// TIA Portal project "MPS_Measuring" (V16)

(* hardware
DEVICE "S7-1200 station_1"  S7-1200 Station
   slot 0: "Rack_0"  S7-1200 Rack  Rack  V1.0
   slot 1: "PLC_1"  CPU 1214C AC/DC/Rly  6ES7 214-1BG40-0XB0  V4.2
DEVICE "S7-1200 station_2"  S7-1200 Station
   slot 0: "Rack_0"  S7-1200 Rack  Rack  V1.0
   slot 1: "PLC_2"  CPU 1214C AC/DC/Rly  6ES7 214-1BG31-0XB0  V3.0
DEVICE "HMI_1"  KTP600 Basic color PN
   slot 0: "HMI_1"  KTP600 Basic color PN  6AV6 647-0AD11-3AX0  12.0.0.0
   slot 1: "HMI_RT_1"  KTP600 Basic color PN  6AV6 647-0AD11-3AX0  12.0.0.0
   slot 5: "HMI_1.IE_CP_1"  PROFINET Interface  12.0.0.0
      slot 1: "PROFINET Interface_1"  PROFINET Interface
         slot 1: "Port_1"  Port
*)

// ===== PLC "PLC_1"  CPU 1214C AC/DC/Rly =====

VAR_GLOBAL   // PLC tag table "Default tag table"
   "Conveyor_fwd" AT %Q0.0 : Bool;
   "Conveyor_rvs" AT %Q0.1 : Bool;
   "Adv_separator" AT %Q0.2 : Bool;
   "Stopper_On" AT %Q0.3 : Bool;
   "Open_Gripper" AT %Q0.4 : Bool;
   "Gripper_dws" AT %Q0.5 : Bool;
   "Swivel_to_msg" AT %Q0.6 : Bool;
   "wp_beg" AT %I0.0 : Bool;
   "wp_mid" AT %I0.1 : Bool;
   "no_wp_end" AT %I0.2 : Bool;
   "Gripper_open" AT %I0.4 : Bool;
   "Gripper_raised" AT %I0.5 : Bool;
   "Swivel_at_conv" AT %I0.6 : Bool;
   "Swivel_at_msg" AT %I0.7 : Bool;
   "Analog_In" AT %IW64 : Int;
   "wp_measure" AT %MD1 : Real;
   "wp_measured" AT %M0.1 : Bool;   // Workpiece has been measured
   "has_cap" AT %M0.2 : Bool;
   "wp_at_conv" AT %M0.3 : Bool;
   "wp_at_msg" AT %M0.4 : Bool;
END_VAR

// folder: System blocks/Program resources

DATA_BLOCK "IEC_Timer_0_DB"   // DB1
{ S7_Optimized_Access := 'TRUE' }
AUTHOR : Simatic
FAMILY : IEC
NAME : IEC_TMR
VERSION : 1.0
// stored: InstanceOfName IEC_TIMER
"IEC_TIMER"
BEGIN
END_DATA_BLOCK

DATA_BLOCK "IEC_Timer_0_DB_1"   // DB2
{ S7_Optimized_Access := 'TRUE' }
AUTHOR : Simatic
FAMILY : IEC
NAME : IEC_TMR
VERSION : 1.0
// stored: InstanceOfName IEC_TIMER
"IEC_TIMER"
BEGIN
END_DATA_BLOCK

DATA_BLOCK "IEC_Timer_0_DB_2"   // DB3
{ S7_Optimized_Access := 'TRUE' }
AUTHOR : Simatic
FAMILY : IEC
NAME : IEC_TMR
VERSION : 1.0
// stored: InstanceOfName IEC_TIMER
"IEC_TIMER"
BEGIN
END_DATA_BLOCK

DATA_BLOCK "IEC_Timer_0_DB_3"   // DB4
{ S7_Optimized_Access := 'TRUE' }
AUTHOR : Simatic
FAMILY : IEC
NAME : IEC_TMR
VERSION : 1.0
// stored: InstanceOfName IEC_TIMER
"IEC_TIMER"
BEGIN
END_DATA_BLOCK

// folder: (top level)

FUNCTION "Read_Analog_Input" : Void   // FC1, LAD
{ S7_Optimized_Access := 'TRUE' }
VERSION : 0.1
   VAR_INPUT
      Input_channel : Int;
      Lower_value : Int;
      Upper_value : Int;
   END_VAR
   VAR_OUTPUT
      Measure : Real;
   END_VAR
   VAR_TEMP
      Temp1 : Real;
   END_VAR
BEGIN

REGION Network 1
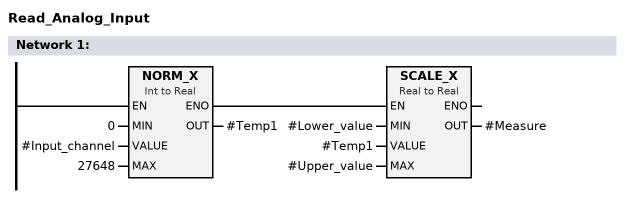
   RUNG wire#powerrail
      { S7_Templates := "[SrcType := Int, DestType := Real]"; S7_GenerateENO := "TRUE" } Normalize(min := 0, value := #Input_channel, max := 27648, out => #Temp1)
      { S7_Templates := "[SrcType := Real, DestType := Real]"; S7_GenerateENO := "TRUE" } Scale(min := #Lower_value, value := #Temp1, max := #Upper_value, out => #Measure)
   END_RUNG
   // the same network as SCL:
   // ENO of a box is taken as its EN; it also drops when the box reports an error
   #Temp1 := NORM_X(MIN := 0, VALUE := #Input_channel, MAX := 27648);
   #Measure := SCALE_X(MIN := #Lower_value, VALUE := #Temp1, MAX := #Upper_value);
END_REGION
END_FUNCTION

FUNCTION "is_capped" : Void   // FC4, LAD
{ S7_Optimized_Access := 'TRUE' }
VERSION : 0.1
   VAR_INPUT
      input_channel : Int;
   END_VAR
   VAR_OUTPUT
      with_cap : Bool;
   END_VAR
   VAR_TEMP
      temp1 : Real;
   END_VAR
   VAR CONSTANT
      cap_det : Real := 0.5;
   END_VAR
   VAR_TEMP   // added for the SCL form of the ladder/FBD networks
      _w1 : Bool;
   END_VAR
BEGIN

REGION Network 1
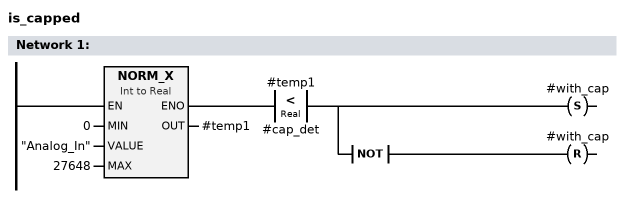
   RUNG wire#powerrail
      { S7_Templates := "[SrcType := Int, DestType := Real]"; S7_GenerateENO := "TRUE" } Normalize(min := 0, value := "Analog_In", max := 27648, out => #temp1)
      { S7_Templates := "SrcType := Real" } LT_Contact(in1 := #temp1, in2 := #cap_det)
      wire#w1
      S_Coil( #with_cap )
   END_RUNG
   RUNG wire#w1
      Not()
      R_Coil( #with_cap )
   END_RUNG
   // the same network as SCL:
   // ENO of a box is taken as its EN; it also drops when the box reports an error
   #temp1 := NORM_X(MIN := 0, VALUE := "Analog_In", MAX := 27648);
   #_w1 := #temp1 < #cap_det;
   IF #_w1 THEN #with_cap := TRUE; END_IF;
   IF NOT #_w1 THEN #with_cap := FALSE; END_IF;
END_REGION
END_FUNCTION

ORGANIZATION_BLOCK "Main"   // OB1, LAD, ProgramCycle
TITLE = "Main Program Sweep (Cycle)"
{ S7_Optimized_Access := 'TRUE' }
VERSION : 0.1
   VAR_TEMP   // added for the SCL form of the ladder/FBD networks
      _w1 : Bool;
   END_VAR
BEGIN

REGION Network 1: Workpiece has been measured
   // Read Measurement
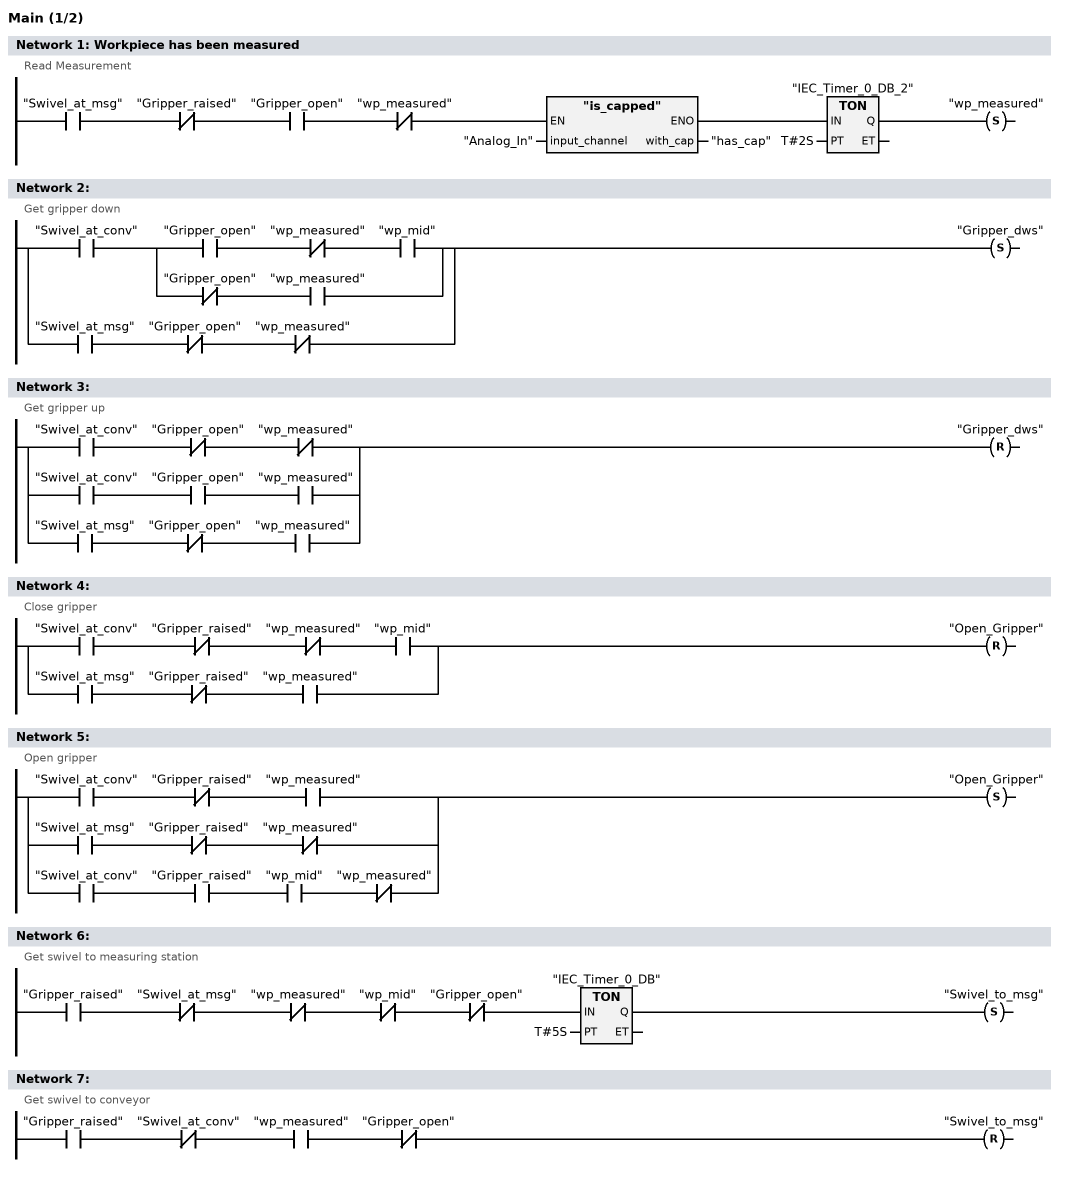
   "is_capped"(EN := "Swivel_at_msg" AND NOT "Gripper_raised" AND "Gripper_open" AND NOT "wp_measured",
               input_channel := "Analog_In",
               with_cap => "has_cap",
               ENO => #_w1);
   "IEC_Timer_0_DB_2".TON(IN := #_w1, PT := T#2S);
   IF "IEC_Timer_0_DB_2".Q THEN "wp_measured" := TRUE; END_IF;
END_REGION

REGION Network 2
   // Get gripper down
   RUNG wire#powerrail
      Contact( "Swivel_at_conv" )
      wire#w1
      Contact( "Gripper_open" )
      I_Contact( "wp_measured" )
      Contact( "wp_mid" )
      wire#w2
      S_Coil( "Gripper_dws" )
   END_RUNG
   RUNG wire#w1
      I_Contact( "Gripper_open" )
      Contact( "wp_measured" )
   END_RUNG wire#w2
   RUNG wire#powerrail
      Contact( "Swivel_at_msg" )
      I_Contact( "Gripper_open" )
      I_Contact( "wp_measured" )
   END_RUNG wire#w2
   // the same network as SCL:
   IF ("Swivel_at_conv" AND (("Gripper_open" AND NOT "wp_measured" AND "wp_mid") OR (NOT "Gripper_open" AND "wp_measured"))) OR ("Swivel_at_msg" AND NOT "Gripper_open" AND NOT "wp_measured") THEN
       "Gripper_dws" := TRUE;
   END_IF;
END_REGION

REGION Network 3
   // Get gripper up
   RUNG wire#powerrail
      Contact( "Swivel_at_conv" )
      I_Contact( "Gripper_open" )
      I_Contact( "wp_measured" )
      wire#w1
      R_Coil( "Gripper_dws" )
   END_RUNG
   RUNG wire#powerrail
      Contact( "Swivel_at_conv" )
      Contact( "Gripper_open" )
      Contact( "wp_measured" )
   END_RUNG wire#w1
   RUNG wire#powerrail
      Contact( "Swivel_at_msg" )
      I_Contact( "Gripper_open" )
      Contact( "wp_measured" )
   END_RUNG wire#w1
   // the same network as SCL:
   IF ("Swivel_at_conv" AND NOT "Gripper_open" AND NOT "wp_measured") OR ("Swivel_at_conv" AND "Gripper_open" AND "wp_measured") OR ("Swivel_at_msg" AND NOT "Gripper_open" AND "wp_measured") THEN
       "Gripper_dws" := FALSE;
   END_IF;
END_REGION

REGION Network 4
   // Close gripper
   RUNG wire#powerrail
      Contact( "Swivel_at_conv" )
      I_Contact( "Gripper_raised" )
      I_Contact( "wp_measured" )
      Contact( "wp_mid" )
      wire#w1
      R_Coil( "Open_Gripper" )
   END_RUNG
   RUNG wire#powerrail
      Contact( "Swivel_at_msg" )
      I_Contact( "Gripper_raised" )
      Contact( "wp_measured" )
   END_RUNG wire#w1
   // the same network as SCL:
   IF ("Swivel_at_conv" AND NOT "Gripper_raised" AND NOT "wp_measured" AND "wp_mid") OR ("Swivel_at_msg" AND NOT "Gripper_raised" AND "wp_measured") THEN
       "Open_Gripper" := FALSE;
   END_IF;
END_REGION

REGION Network 5
   // Open gripper
   RUNG wire#powerrail
      Contact( "Swivel_at_conv" )
      I_Contact( "Gripper_raised" )
      Contact( "wp_measured" )
      wire#w1
      S_Coil( "Open_Gripper" )
   END_RUNG
   RUNG wire#powerrail
      Contact( "Swivel_at_msg" )
      I_Contact( "Gripper_raised" )
      I_Contact( "wp_measured" )
   END_RUNG wire#w1
   RUNG wire#powerrail
      Contact( "Swivel_at_conv" )
      Contact( "Gripper_raised" )
      Contact( "wp_mid" )
      I_Contact( "wp_measured" )
   END_RUNG wire#w1
   // the same network as SCL:
   IF ("Swivel_at_conv" AND NOT "Gripper_raised" AND "wp_measured") OR ("Swivel_at_msg" AND NOT "Gripper_raised" AND NOT "wp_measured") OR ("Swivel_at_conv" AND "Gripper_raised" AND "wp_mid" AND NOT "wp_measured") THEN
       "Open_Gripper" := TRUE;
   END_IF;
END_REGION

REGION Network 6
   // Get swivel to measuring station
   "IEC_Timer_0_DB".TON(IN := "Gripper_raised" AND NOT "Swivel_at_msg" AND NOT "wp_measured" AND NOT "wp_mid" AND NOT "Gripper_open",
                        PT := T#5S);
   IF "IEC_Timer_0_DB".Q THEN "Swivel_to_msg" := TRUE; END_IF;
END_REGION

REGION Network 7
   // Get swivel to conveyor
   RUNG wire#powerrail
      Contact( "Gripper_raised" )
      I_Contact( "Swivel_at_conv" )
      Contact( "wp_measured" )
      I_Contact( "Gripper_open" )
      R_Coil( "Swivel_to_msg" )
   END_RUNG
   // the same network as SCL:
   IF "Gripper_raised" AND NOT "Swivel_at_conv" AND "wp_measured" AND NOT "Gripper_open" THEN
       "Swivel_to_msg" := FALSE;
   END_IF;
END_REGION

REGION Network 8
   // Advance separator
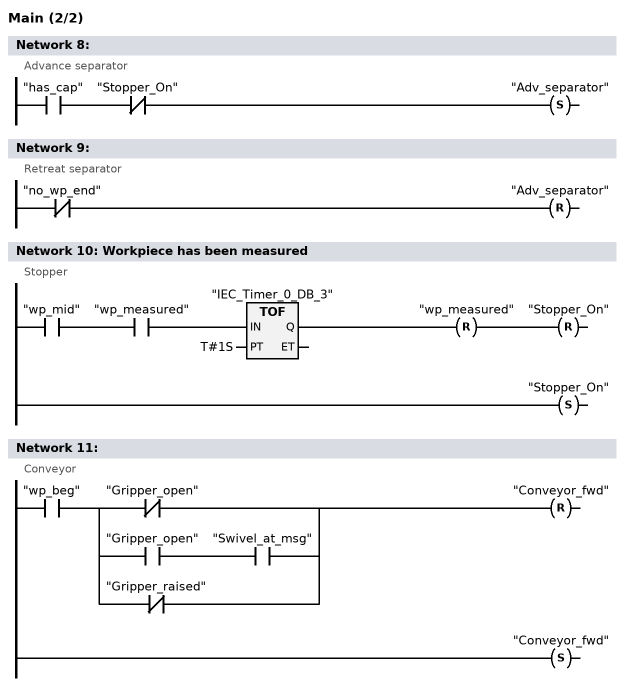
   RUNG wire#powerrail
      Contact( "has_cap" )
      I_Contact( "Stopper_On" )
      S_Coil( "Adv_separator" )
   END_RUNG
   // the same network as SCL:
   IF "has_cap" AND NOT "Stopper_On" THEN "Adv_separator" := TRUE; END_IF;
END_REGION

REGION Network 9
   // Retreat separator
   RUNG wire#powerrail
      I_Contact( "no_wp_end" )
      R_Coil( "Adv_separator" )
   END_RUNG
   // the same network as SCL:
   IF NOT "no_wp_end" THEN "Adv_separator" := FALSE; END_IF;
END_REGION

REGION Network 10: Workpiece has been measured
   // Stopper
   "IEC_Timer_0_DB_3".TOF(IN := "wp_mid" AND "wp_measured", PT := T#1S);
   IF "IEC_Timer_0_DB_3".Q THEN
       "wp_measured" := FALSE;
       "Stopper_On" := FALSE;
   END_IF;
   "Stopper_On" := TRUE;
END_REGION

REGION Network 11
   // Conveyor
   RUNG wire#powerrail
      Contact( "wp_beg" )
      wire#w1
      I_Contact( "Gripper_open" )
      wire#w2
      R_Coil( "Conveyor_fwd" )
   END_RUNG
   RUNG wire#w1
      Contact( "Gripper_open" )
      Contact( "Swivel_at_msg" )
   END_RUNG wire#w2
   RUNG wire#w1
      I_Contact( "Gripper_raised" )
   END_RUNG wire#w2
   RUNG wire#powerrail
      S_Coil( "Conveyor_fwd" )
   END_RUNG
   // the same network as SCL:
   IF "wp_beg" AND (NOT "Gripper_open" OR ("Gripper_open" AND "Swivel_at_msg") OR NOT "Gripper_raised") THEN
       "Conveyor_fwd" := FALSE;
   END_IF;
   "Conveyor_fwd" := TRUE;
END_REGION
END_ORGANIZATION_BLOCK

ORGANIZATION_BLOCK "Startup"   // OB100, LAD, Startup
TITLE = "Complete Restart"
{ S7_Optimized_Access := 'TRUE' }
VERSION : 0.1
   VAR_INPUT
      LostRetentive : Bool;   // True if retentive data are lost
      LostRTC : Bool;   // True if date and time are lost
   END_VAR
BEGIN

REGION Network 1
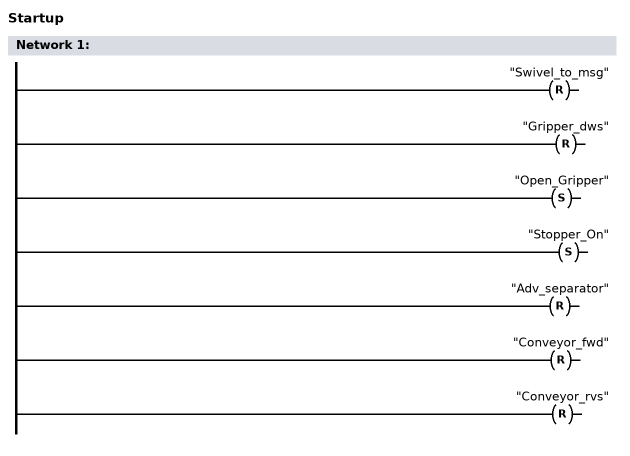
   RUNG wire#powerrail
      R_Coil( "Swivel_to_msg" )
   END_RUNG
   RUNG wire#powerrail
      R_Coil( "Gripper_dws" )
   END_RUNG
   RUNG wire#powerrail
      S_Coil( "Open_Gripper" )
   END_RUNG
   RUNG wire#powerrail
      S_Coil( "Stopper_On" )
   END_RUNG
   RUNG wire#powerrail
      R_Coil( "Adv_separator" )
   END_RUNG
   RUNG wire#powerrail
      R_Coil( "Conveyor_fwd" )
   END_RUNG
   RUNG wire#powerrail
      R_Coil( "Conveyor_rvs" )
   END_RUNG
   // the same network as SCL:
   "Swivel_to_msg" := FALSE;
   "Gripper_dws" := FALSE;
   "Open_Gripper" := TRUE;
   "Stopper_On" := TRUE;
   "Adv_separator" := FALSE;
   "Conveyor_fwd" := FALSE;
   "Conveyor_rvs" := FALSE;
END_REGION
END_ORGANIZATION_BLOCK

// ===== PLC "PLC_2"  CPU 1214C AC/DC/Rly =====

VAR_GLOBAL   // PLC tag table "Default tag table_1"
   "Conveyor_fwd" AT %Q0.0 : Bool;
   "Conveyor_rvs" AT %Q0.1 : Bool;
   "Adv_separator" AT %Q0.2 : Bool;
   "Retract_stopper" AT %Q0.3 : Bool;
   "Open_Gripper" AT %Q0.4 : Bool;
   "Gripper_dws" AT %Q0.5 : Bool;
   "Swivel_to_msg" AT %Q0.6 : Bool;
   "wp_beg" AT %I0.0 : Bool;
   "wp_mid" AT %I0.1 : Bool;
   "no_wp_end" AT %I0.2 : Bool;
   "Gripper_open" AT %I0.6 : Bool;
   "Gripper_raised" AT %I0.5 : Bool;
   "Swivel_at_conv" AT %I0.4 : Bool;
   "Swivel_at_msg" AT %I0.7 : Bool;
   "Analog_In" AT %IW64 : Int;
   "wp_measure" AT %MD1 : Real;
   "wp_measured" AT %M0.1 : Bool;   // Workpiece has been measured
   "has_cap" AT %M0.2 : Bool;
   "wp_at_conv" AT %M0.3 : Bool;
   "wp_at_msg" AT %M0.4 : Bool;
   "stopper_shall_retract" AT %M0.5 : Bool;
   "conv_shall_adv" AT %M0.6 : Bool;
   "system_ready" AT %M0.7 : Bool;
   "reset" AT %M5.0 : Bool;
END_VAR

VAR_GLOBAL CONSTANT   // PLC tag table "Default tag table_1"
   "Local~PROFINET_interface_1~Port_1(1)" : Hw_Interface := 65;
   "OB_Main(1)" : OB_PCYCLE := 1;
   "OB_Startup" : OB_STARTUP := 100;
   "Local(1)" : Hw_SubModule := 49;
   "Local~DI_14_DQ_10_1(1)" : Hw_SubModule := 264;
   "Local~AI_2_1(1)" : Hw_SubModule := 263;
   "Local~MC" : Hw_SubModule := 51;
   "Local~Common" : Hw_SubModule := 50;
   "Local~Device" : Hw_Device := 32;
   "Local~Configuration" : Hw_SubModule := 33;
   "Local~Exec" : Hw_SubModule := 52;
   "Local~HSC_1(1)" : Hw_Hsc := 257;
   "Local~HSC_2(1)" : Hw_Hsc := 258;
   "Local~HSC_3(1)" : Hw_Hsc := 259;
   "Local~HSC_4(1)" : Hw_Hsc := 260;
   "Local~HSC_5(1)" : Hw_Hsc := 261;
   "Local~HSC_6(1)" : Hw_Hsc := 262;
   "Local~Pulse_1(1)" : Hw_Pwm := 265;
   "Local~Pulse_2(1)" : Hw_Pwm := 266;
   "Local~Pulse_3(1)" : Hw_Pwm := 267;
   "Local~Pulse_4(1)" : Hw_Pwm := 268;
   "Local~PROFINET_interface_1(1)" : Hw_Interface := 64;
   "None" : Pip := 65535;
   "Automatic update" : Pip := 0;
   "PIP 1" : Pip := 1;
   "PIP 2" : Pip := 2;
   "PIP 3" : Pip := 3;
   "PIP 4" : Pip := 4;
   "PIP OB Servo" : Pip := 32768;
END_VAR

// folder: System blocks/Program resources

DATA_BLOCK "IEC_Timer_0_DB"   // DB1
{ S7_Optimized_Access := 'TRUE' }
AUTHOR : Simatic
FAMILY : IEC
NAME : IEC_TMR
VERSION : 1.0
// stored: InstanceOfName IEC_TIMER
"IEC_TIMER"
BEGIN
END_DATA_BLOCK

DATA_BLOCK "IEC_Timer_0_DB_1"   // DB2
{ S7_Optimized_Access := 'TRUE' }
AUTHOR : Simatic
FAMILY : IEC
NAME : IEC_TMR
VERSION : 1.0
// stored: InstanceOfName IEC_TIMER
"IEC_TIMER"
BEGIN
END_DATA_BLOCK

DATA_BLOCK "IEC_Timer_0_DB_2"   // DB3
{ S7_Optimized_Access := 'TRUE' }
AUTHOR : Simatic
FAMILY : IEC
NAME : IEC_TMR
VERSION : 1.0
// stored: InstanceOfName IEC_TIMER
"IEC_TIMER"
BEGIN
END_DATA_BLOCK

DATA_BLOCK "IEC_Timer_0_DB_3"   // DB4
{ S7_Optimized_Access := 'TRUE' }
AUTHOR : Simatic
FAMILY : IEC
NAME : IEC_TMR
VERSION : 1.0
// stored: InstanceOfName IEC_TIMER
"IEC_TIMER"
BEGIN
END_DATA_BLOCK

DATA_BLOCK "IEC_Timer_0_DB_4"   // DB5
{ S7_Optimized_Access := 'TRUE' }
AUTHOR : Simatic
FAMILY : IEC
NAME : IEC_TMR
VERSION : 1.0
// stored: InstanceOfName IEC_TIMER
"IEC_TIMER"
BEGIN
END_DATA_BLOCK

DATA_BLOCK "IEC_Timer_0_DB_5"   // DB6
{ S7_Optimized_Access := 'TRUE' }
AUTHOR : Simatic
FAMILY : IEC
NAME : IEC_TMR
VERSION : 1.0
// stored: InstanceOfName IEC_TIMER
"IEC_TIMER"
BEGIN
END_DATA_BLOCK

DATA_BLOCK "IEC_Timer_0_DB_6"   // DB7
{ S7_Optimized_Access := 'TRUE' }
AUTHOR : Simatic
FAMILY : IEC
NAME : IEC_TMR
VERSION : 1.0
// stored: InstanceOfName IEC_TIMER
"IEC_TIMER"
BEGIN
END_DATA_BLOCK

DATA_BLOCK "IEC_Timer_0_DB_7"   // DB8
{ S7_Optimized_Access := 'TRUE' }
AUTHOR : Simatic
FAMILY : IEC
NAME : IEC_TMR
VERSION : 1.0
// stored: InstanceOfName IEC_TIMER
"IEC_TIMER"
BEGIN
END_DATA_BLOCK

DATA_BLOCK "IEC_Timer_0_DB_8"   // DB9
{ S7_Optimized_Access := 'TRUE' }
AUTHOR : Simatic
FAMILY : IEC
NAME : IEC_TMR
VERSION : 1.0
// stored: InstanceOfName IEC_TIMER
"IEC_TIMER"
BEGIN
END_DATA_BLOCK

DATA_BLOCK "IEC_Timer_0_DB_9"   // DB10
{ S7_Optimized_Access := 'TRUE' }
AUTHOR : Simatic
FAMILY : IEC
NAME : IEC_TMR
VERSION : 1.0
// stored: InstanceOfName IEC_TIMER
"IEC_TIMER"
BEGIN
END_DATA_BLOCK

// folder: (top level)

FUNCTION "reset_block" : Void   // FC1, LAD
{ S7_Optimized_Access := 'TRUE' }
VERSION : 0.1
BEGIN

REGION Network 1
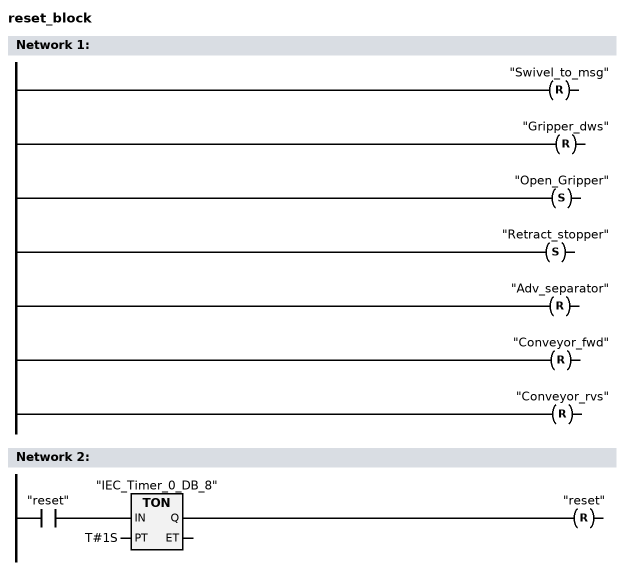
   RUNG wire#powerrail
      R_Coil( "Swivel_to_msg" )
   END_RUNG
   RUNG wire#powerrail
      R_Coil( "Gripper_dws" )
   END_RUNG
   RUNG wire#powerrail
      S_Coil( "Open_Gripper" )
   END_RUNG
   RUNG wire#powerrail
      S_Coil( "Retract_stopper" )
   END_RUNG
   RUNG wire#powerrail
      R_Coil( "Adv_separator" )
   END_RUNG
   RUNG wire#powerrail
      R_Coil( "Conveyor_fwd" )
   END_RUNG
   RUNG wire#powerrail
      R_Coil( "Conveyor_rvs" )
   END_RUNG
   // the same network as SCL:
   "Swivel_to_msg" := FALSE;
   "Gripper_dws" := FALSE;
   "Open_Gripper" := TRUE;
   "Retract_stopper" := TRUE;
   "Adv_separator" := FALSE;
   "Conveyor_fwd" := FALSE;
   "Conveyor_rvs" := FALSE;
END_REGION

REGION Network 2
   "IEC_Timer_0_DB_8".TON(IN := "reset", PT := T#1S);
   IF "IEC_Timer_0_DB_8".Q THEN "reset" := FALSE; END_IF;
END_REGION
END_FUNCTION

FUNCTION "is_capped" : Void   // FC4, LAD
{ S7_Optimized_Access := 'TRUE' }
VERSION : 0.1
   VAR_INPUT
      input_channel : Int;
   END_VAR
   VAR_OUTPUT
      with_cap : Bool;
   END_VAR
   VAR_TEMP
      temp1 : Real;
   END_VAR
   VAR CONSTANT
      cap_det : Real := 0.2;
   END_VAR
   VAR_TEMP   // added for the SCL form of the ladder/FBD networks
      _w1 : Bool;
   END_VAR
BEGIN

REGION Network 1
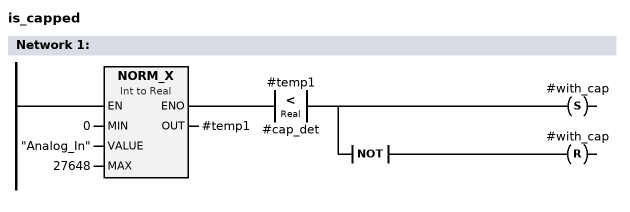
   RUNG wire#powerrail
      { S7_Templates := "[SrcType := Int, DestType := Real]"; S7_GenerateENO := "TRUE" } Normalize(min := 0, value := "Analog_In", max := 27648, out => #temp1)
      { S7_Templates := "SrcType := Real" } LT_Contact(in1 := #temp1, in2 := #cap_det)
      wire#w1
      S_Coil( #with_cap )
   END_RUNG
   RUNG wire#w1
      Not()
      R_Coil( #with_cap )
   END_RUNG
   // the same network as SCL:
   // ENO of a box is taken as its EN; it also drops when the box reports an error
   #temp1 := NORM_X(MIN := 0, VALUE := "Analog_In", MAX := 27648);
   #_w1 := #temp1 < #cap_det;
   IF #_w1 THEN #with_cap := TRUE; END_IF;
   IF NOT #_w1 THEN #with_cap := FALSE; END_IF;
END_REGION
END_FUNCTION

ORGANIZATION_BLOCK "Main"   // OB1, LAD, ProgramCycle
TITLE = "Main Program Sweep (Cycle)"
{ S7_Optimized_Access := 'TRUE' }
VERSION : 0.1
   VAR_TEMP   // added for the SCL form of the ladder/FBD networks
      _w1 : Bool;
      _w2 : Bool;
   END_VAR
BEGIN

REGION Network 1: Workpiece has been measured
   // Read Measurement
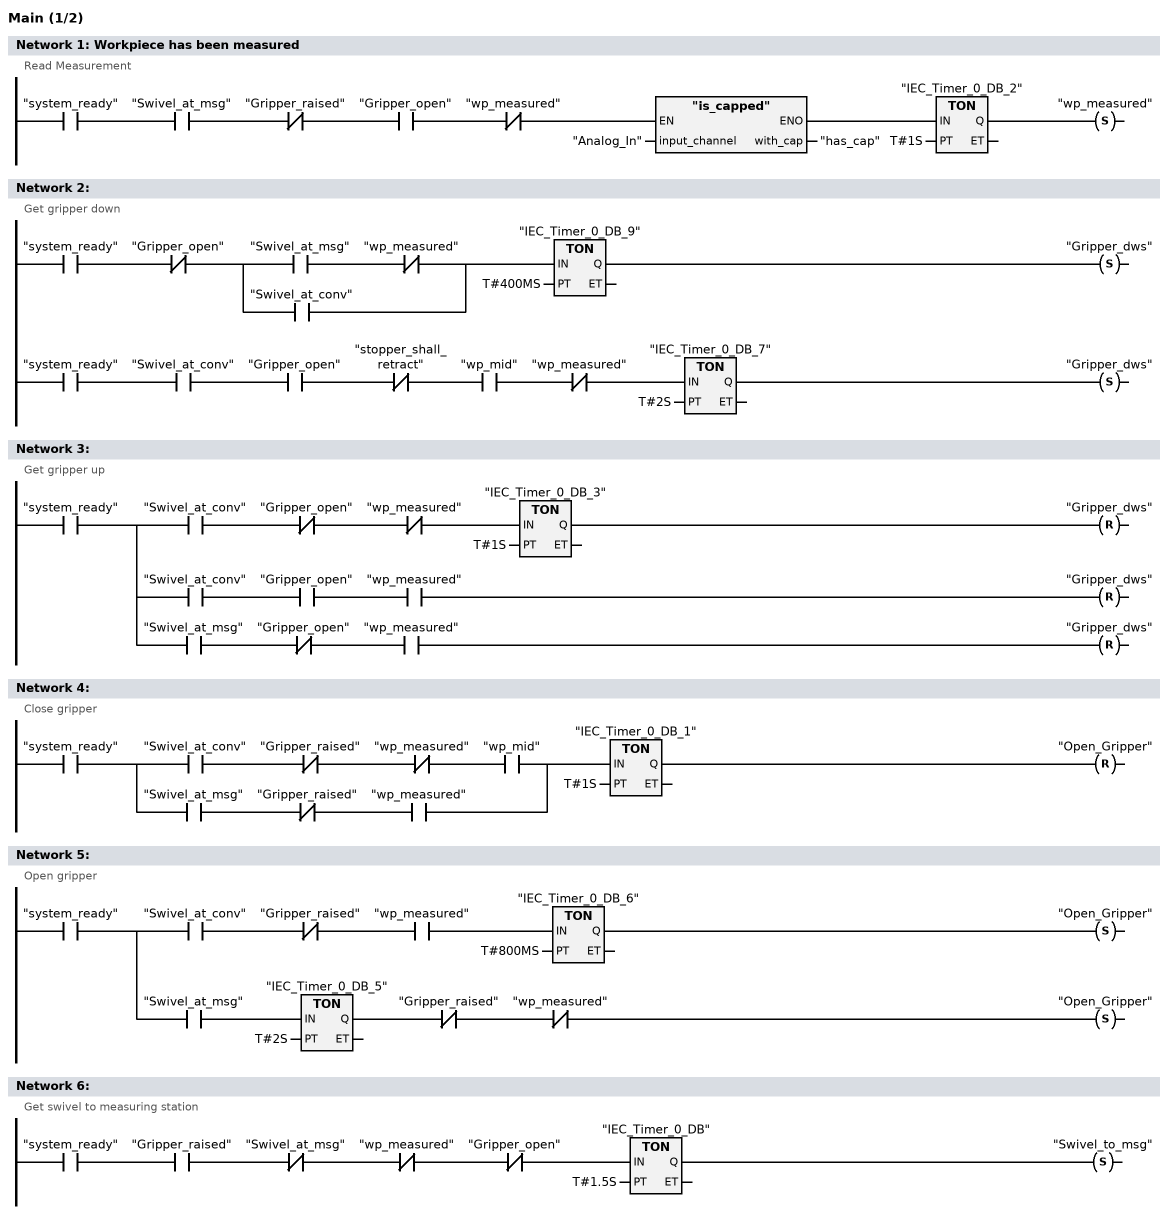
   "is_capped"(EN := "system_ready" AND "Swivel_at_msg" AND NOT "Gripper_raised" AND "Gripper_open" AND NOT "wp_measured",
               input_channel := "Analog_In",
               with_cap => "has_cap",
               ENO => #_w1);
   "IEC_Timer_0_DB_2".TON(IN := #_w1, PT := T#1S);
   IF "IEC_Timer_0_DB_2".Q THEN "wp_measured" := TRUE; END_IF;
END_REGION

REGION Network 2
   // Get gripper down
   "IEC_Timer_0_DB_9".TON(IN := "system_ready" AND NOT "Gripper_open" AND (("Swivel_at_msg" AND NOT "wp_measured") OR "Swivel_at_conv"),
                          PT := T#400MS);
   IF "IEC_Timer_0_DB_9".Q THEN "Gripper_dws" := TRUE; END_IF;
   "IEC_Timer_0_DB_7".TON(IN := "system_ready" AND "Swivel_at_conv" AND "Gripper_open" AND NOT "stopper_shall_retract" AND "wp_mid" AND NOT "wp_measured",
                          PT := T#2S);
   IF "IEC_Timer_0_DB_7".Q THEN "Gripper_dws" := TRUE; END_IF;
END_REGION

REGION Network 3
   // Get gripper up
   "IEC_Timer_0_DB_3".TON(IN := "system_ready" AND "Swivel_at_conv" AND NOT "Gripper_open" AND NOT "wp_measured",
                          PT := T#1S);
   IF "IEC_Timer_0_DB_3".Q THEN "Gripper_dws" := FALSE; END_IF;
   IF "system_ready" AND "Swivel_at_conv" AND "Gripper_open" AND "wp_measured" THEN
       "Gripper_dws" := FALSE;
   END_IF;
   IF "system_ready" AND "Swivel_at_msg" AND NOT "Gripper_open" AND "wp_measured" THEN
       "Gripper_dws" := FALSE;
   END_IF;
END_REGION

REGION Network 4
   // Close gripper
   "IEC_Timer_0_DB_1".TON(IN := "system_ready" AND (("Swivel_at_conv" AND NOT "Gripper_raised" AND NOT "wp_measured" AND "wp_mid") OR ("Swivel_at_msg" AND NOT "Gripper_raised" AND "wp_measured")),
                          PT := T#1S);
   IF "IEC_Timer_0_DB_1".Q THEN "Open_Gripper" := FALSE; END_IF;
END_REGION

REGION Network 5
   // Open gripper
   "IEC_Timer_0_DB_6".TON(IN := "system_ready" AND "Swivel_at_conv" AND NOT "Gripper_raised" AND "wp_measured",
                          PT := T#800MS);
   IF "IEC_Timer_0_DB_6".Q THEN "Open_Gripper" := TRUE; END_IF;
   "IEC_Timer_0_DB_5".TON(IN := "system_ready" AND "Swivel_at_msg", PT := T#2S);
   IF "IEC_Timer_0_DB_5".Q AND NOT "Gripper_raised" AND NOT "wp_measured" THEN
       "Open_Gripper" := TRUE;
   END_IF;
END_REGION

REGION Network 6
   // Get swivel to measuring station
   "IEC_Timer_0_DB".TON(IN := "system_ready" AND "Gripper_raised" AND NOT "Swivel_at_msg" AND NOT "wp_measured" AND NOT "Gripper_open",
                        PT := T#1.5S);
   IF "IEC_Timer_0_DB".Q THEN "Swivel_to_msg" := TRUE; END_IF;
END_REGION

REGION Network 7
   // Get swivel to conveyor
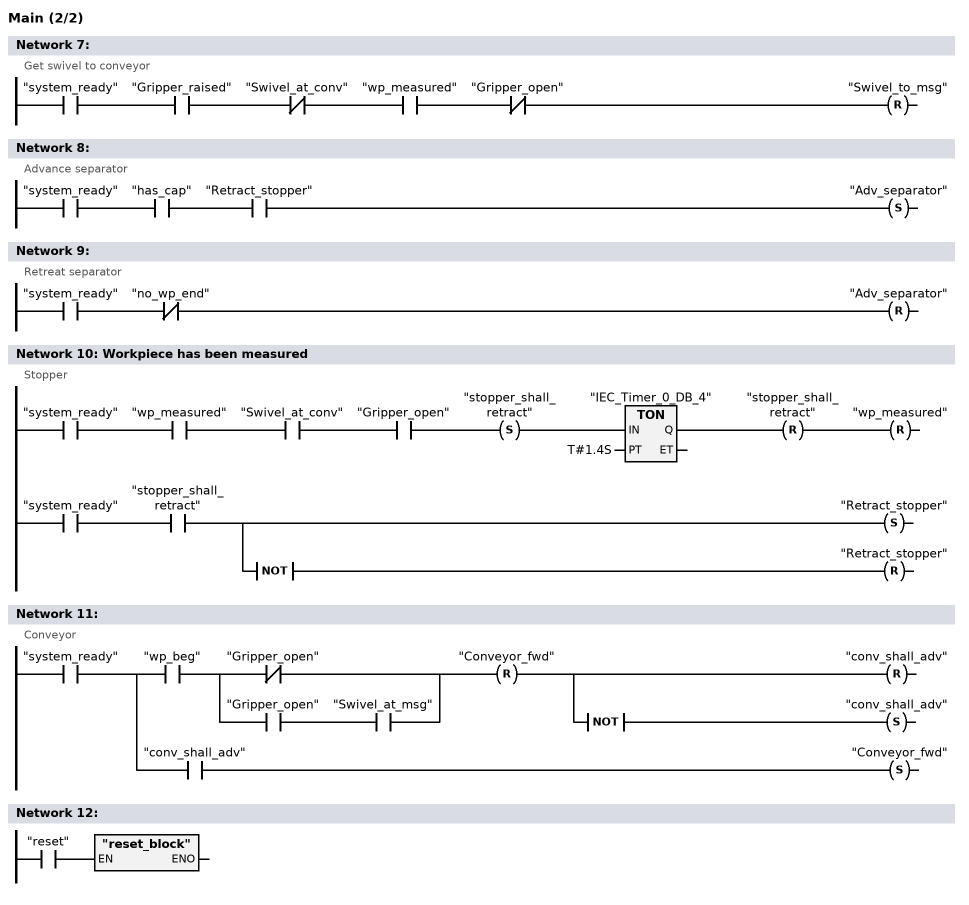
   RUNG wire#powerrail
      Contact( "system_ready" )
      Contact( "Gripper_raised" )
      I_Contact( "Swivel_at_conv" )
      Contact( "wp_measured" )
      I_Contact( "Gripper_open" )
      R_Coil( "Swivel_to_msg" )
   END_RUNG
   // the same network as SCL:
   IF "system_ready" AND "Gripper_raised" AND NOT "Swivel_at_conv" AND "wp_measured" AND NOT "Gripper_open" THEN
       "Swivel_to_msg" := FALSE;
   END_IF;
END_REGION

REGION Network 8
   // Advance separator
   RUNG wire#powerrail
      Contact( "system_ready" )
      Contact( "has_cap" )
      Contact( "Retract_stopper" )
      S_Coil( "Adv_separator" )
   END_RUNG
   // the same network as SCL:
   IF "system_ready" AND "has_cap" AND "Retract_stopper" THEN "Adv_separator" := TRUE; END_IF;
END_REGION

REGION Network 9
   // Retreat separator
   RUNG wire#powerrail
      Contact( "system_ready" )
      I_Contact( "no_wp_end" )
      R_Coil( "Adv_separator" )
   END_RUNG
   // the same network as SCL:
   IF "system_ready" AND NOT "no_wp_end" THEN "Adv_separator" := FALSE; END_IF;
END_REGION

REGION Network 10: Workpiece has been measured
   // Stopper
   #_w1 := "system_ready" AND "wp_measured" AND "Swivel_at_conv" AND "Gripper_open";
   IF #_w1 THEN "stopper_shall_retract" := TRUE; END_IF;
   "IEC_Timer_0_DB_4".TON(IN := #_w1, PT := T#1.4S);
   IF "IEC_Timer_0_DB_4".Q THEN
       "stopper_shall_retract" := FALSE;
       "wp_measured" := FALSE;
   END_IF;
   #_w2 := "system_ready" AND "stopper_shall_retract";
   IF #_w2 THEN "Retract_stopper" := TRUE; END_IF;
   IF NOT #_w2 THEN "Retract_stopper" := FALSE; END_IF;
END_REGION

REGION Network 11
   // Conveyor
   RUNG wire#powerrail
      Contact( "system_ready" )
      wire#w1
      Contact( "wp_beg" )
      wire#w2
      I_Contact( "Gripper_open" )
      wire#w3
      R_Coil( "Conveyor_fwd" )
      wire#w4
      R_Coil( "conv_shall_adv" )
   END_RUNG
   RUNG wire#w2
      Contact( "Gripper_open" )
      Contact( "Swivel_at_msg" )
   END_RUNG wire#w3
   RUNG wire#w4
      Not()
      S_Coil( "conv_shall_adv" )
   END_RUNG
   RUNG wire#w1
      Contact( "conv_shall_adv" )
      S_Coil( "Conveyor_fwd" )
   END_RUNG
   // the same network as SCL:
   #_w1 := "system_ready" AND "wp_beg" AND (NOT "Gripper_open" OR ("Gripper_open" AND "Swivel_at_msg"));
   IF #_w1 THEN
       "Conveyor_fwd" := FALSE;
       "conv_shall_adv" := FALSE;
   END_IF;
   IF NOT #_w1 THEN "conv_shall_adv" := TRUE; END_IF;
   IF "system_ready" AND "conv_shall_adv" THEN "Conveyor_fwd" := TRUE; END_IF;
END_REGION

REGION Network 12
   RUNG wire#powerrail
      Contact( "reset" )
      "reset_block"()
   END_RUNG
   // the same network as SCL:
   IF "reset" THEN "reset_block"(); END_IF;
END_REGION
END_ORGANIZATION_BLOCK

ORGANIZATION_BLOCK "Startup"   // OB100, LAD, Startup
TITLE = "Complete Restart"
{ S7_Optimized_Access := 'TRUE' }
VERSION : 0.1
   VAR_INPUT
      LostRetentive : Bool;   // True if retentive data are lost
      LostRTC : Bool;   // True if date and time are lost
   END_VAR
BEGIN

REGION Network 1
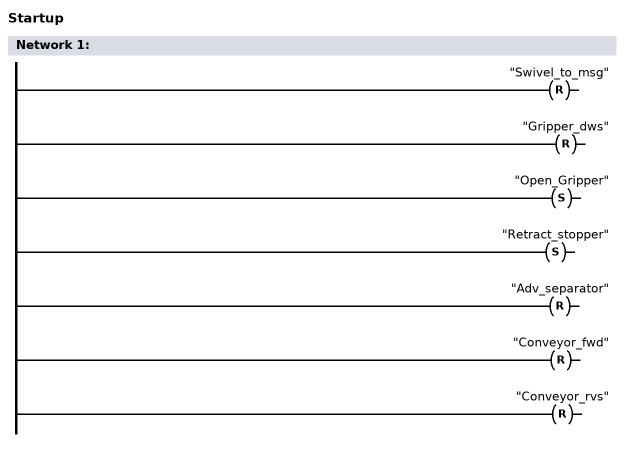
   RUNG wire#powerrail
      R_Coil( "Swivel_to_msg" )
   END_RUNG
   RUNG wire#powerrail
      R_Coil( "Gripper_dws" )
   END_RUNG
   RUNG wire#powerrail
      S_Coil( "Open_Gripper" )
   END_RUNG
   RUNG wire#powerrail
      S_Coil( "Retract_stopper" )
   END_RUNG
   RUNG wire#powerrail
      R_Coil( "Adv_separator" )
   END_RUNG
   RUNG wire#powerrail
      R_Coil( "Conveyor_fwd" )
   END_RUNG
   RUNG wire#powerrail
      R_Coil( "Conveyor_rvs" )
   END_RUNG
   // the same network as SCL:
   "Swivel_to_msg" := FALSE;
   "Gripper_dws" := FALSE;
   "Open_Gripper" := TRUE;
   "Retract_stopper" := TRUE;
   "Adv_separator" := FALSE;
   "Conveyor_fwd" := FALSE;
   "Conveyor_rvs" := FALSE;
END_REGION
END_ORGANIZATION_BLOCK

(* ===== HMI "HMI_RT_1" =====
system functions are stored by id; their names below are inferred from use
connection "HMI_Connection_1": ETHERNET, SMART_S7_1200_OMS

HMI tags "Default tag table"
   "Tag_ScreenNumber" : UInt, internal
   "system_ready" : Bool = PLC system_ready AT %M0.7, 1 s
   "reset" : Bool = PLC reset AT %M5.0, 1 s

Template "Template_1" 320x240
   Button "Exit" at 266,202 size 52x37; TextOff 'Exit'; PictureOff "ExitRuntime_KTP600_Basic_color_PN"; PictureOn "ExitRuntime_KTP600_Basic_color_PN"
      on Release: StopRuntime(0)
   Button "Template_Button" at 213,202 size 52x37; TextOff 'Text'
   Button "Template_Button_1" at 160,202 size 52x37; TextOff 'Text'
   Button "Template_Button_2" at 107,202 size 52x37; TextOff 'Text'
   Button "Template_Button_3" at 54,202 size 52x37; TextOff 'Text'
   Button "Start screen" at 1,202 size 52x37; TextOff 'Start screen'; PictureOff "NavigateHome_KTP600_Basic_color_PN"; PictureOn "NavigateHome_KTP600_Basic_color_PN"
      on Release: ActivateScreen("Root screen", 0)
   SymbolicIOField "Symbolic_IO_Field_Screen" at 69,7 size 164x24; TextOff '0'; TextOn '1'; TextList "TextList_ScreenNames"
      ProcessValue <- "Tag_ScreenNumber"
      on Change: ActivateScreenByNumber("Tag_ScreenNumber", 0)
   DateTimeField "HmiScreenItemData" at 235,19 size 85x19
   DateTimeField "HmiScreenItemData_1" at 235,0 size 85x19
   GraphicView "Logo" at 0,0 size 67x38; Picture "Logo of HMI_1"

screen "Root screen" 320x240, template "Template_1"
   on GenerateScreen: SetTag("Tag_ScreenNumber", 1)
   Switch "Switch_1" at 116,70 size 64x32; CaptionText 'Switch'; TextOff 'OFF'; TextOn 'ON'
      ProcessValue <- "system_ready"
   TextField "Text field_1" at 116,39 size 72x25; Text 'System'
   Button "Button_1" at 102,156 size 96x32; TextOff 'RESET'
      on Press: SetBit("reset")
*)